SUBAPPLICATION Uebung_038 (* Lauflicht 8 reine Zeitsteuerung *)
  (* Standard: 61499-2; Description: Copyright (c) 2023 Meisterschulen am Ostbahnhof This program and the accompanying materials are made available under the terms of the Eclipse Public License 2.0 which is available at https://www.eclipse.org/legal/epl-2.0/ SPDX-License-Identifier: EPL-2.0 *)
  (* Version 1.0, 2023-10-23, Franz Höpfinger, Meisterschulen am Ostbahnhof *)
  PACKAGE Uebungen;
  IMPORT Uebungen::const::UT::DefaultPool::OutputNumber_N1;
  IMPORT logiBUS::io::DI::logiBUS_DI::Input_I1;
  IMPORT logiBUS::io::DI::logiBUS_DI::Input_I4;
  IMPORT logiBUS::io::DI::logiBUS_DI_Events::BUTTON_SINGLE_CLICK;
  IMPORT logiBUS::io::DQ::logiBUS_DO::Output_Q1;
  IMPORT logiBUS::io::DQ::logiBUS_DO::Output_Q2;
  IMPORT logiBUS::io::DQ::logiBUS_DO::Output_Q3;
  IMPORT logiBUS::io::DQ::logiBUS_DO::Output_Q4;
  IMPORT logiBUS::io::DQ::logiBUS_DO::Output_Q5;
  IMPORT logiBUS::io::DQ::logiBUS_DO::Output_Q6;
  IMPORT logiBUS::io::DQ::logiBUS_DO::Output_Q7;
  IMPORT logiBUS::io::DQ::logiBUS_DO::Output_Q8;
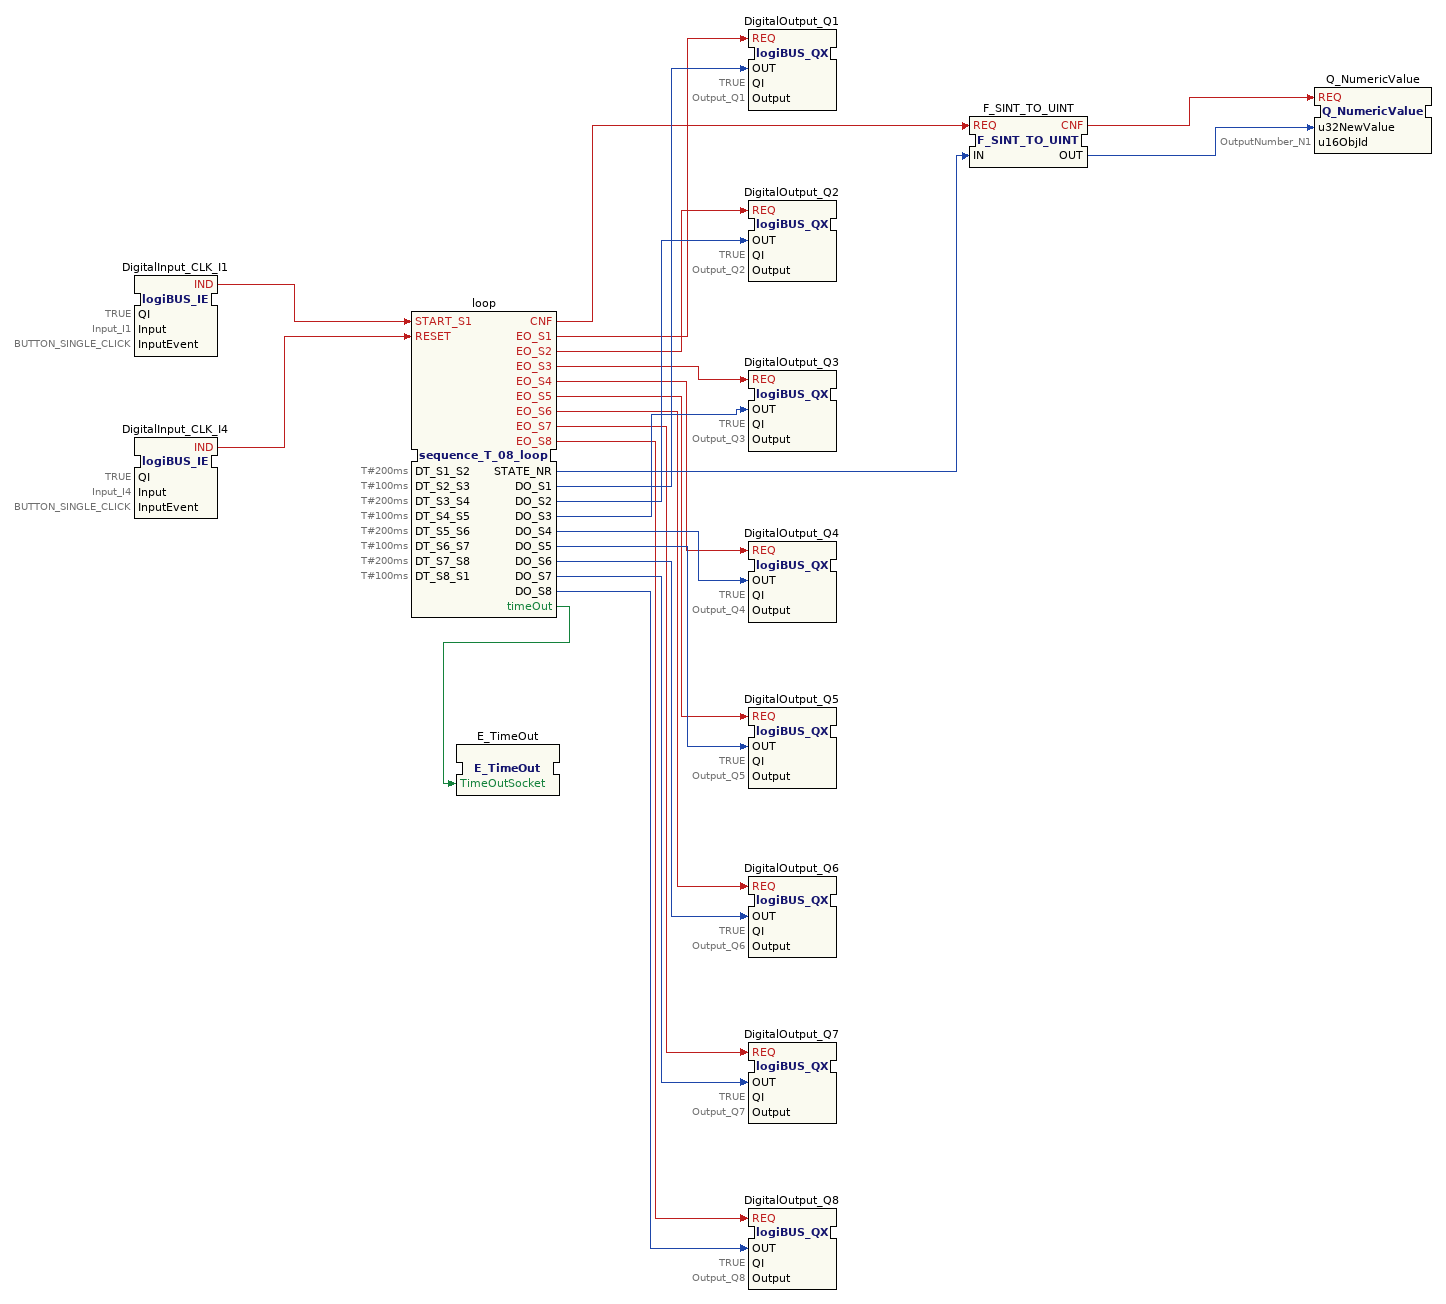
  FBS
    DigitalOutput_Q1 : logiBUS::io::DQ::logiBUS_QX(QI := TRUE, Output := Output_Q1);
    E_TimeOut : iec61499::events::E_TimeOut;
    DigitalOutput_Q2 : logiBUS::io::DQ::logiBUS_QX(QI := TRUE, Output := Output_Q2);
    DigitalOutput_Q3 : logiBUS::io::DQ::logiBUS_QX(QI := TRUE, Output := Output_Q3);
    DigitalOutput_Q4 : logiBUS::io::DQ::logiBUS_QX(QI := TRUE, Output := Output_Q4);
    DigitalInput_CLK_I1 : logiBUS::io::DI::logiBUS_IE(QI := TRUE, Input := Input_I1, InputEvent := BUTTON_SINGLE_CLICK);
    DigitalInput_CLK_I4 : logiBUS::io::DI::logiBUS_IE(QI := TRUE, Input := Input_I4, InputEvent := BUTTON_SINGLE_CLICK);
    DigitalOutput_Q5 : logiBUS::io::DQ::logiBUS_QX(QI := TRUE, Output := Output_Q5);
    DigitalOutput_Q6 : logiBUS::io::DQ::logiBUS_QX(QI := TRUE, Output := Output_Q6);
    DigitalOutput_Q7 : logiBUS::io::DQ::logiBUS_QX(QI := TRUE, Output := Output_Q7);
    DigitalOutput_Q8 : logiBUS::io::DQ::logiBUS_QX(QI := TRUE, Output := Output_Q8);
    Q_NumericValue : isobus::UT::Q::Q_NumericValue(u16ObjId := OutputNumber_N1);
    F_SINT_TO_UINT : iec61131::conversion::F_SINT_TO_UINT;
    loop : logiBUS::utils::sequence::timed::sequence_T_08_loop(DT_S1_S2 := T#200ms, DT_S2_S3 := T#100ms, DT_S3_S4 := T#200ms, DT_S4_S5 := T#100ms, DT_S5_S6 := T#200ms, DT_S6_S7 := T#100ms, DT_S7_S8 := T#200ms, DT_S8_S1 := T#100ms);
  END_FBS
  EVENT_CONNECTIONS
    F_SINT_TO_UINT.CNF TO Q_NumericValue.REQ;
    DigitalInput_CLK_I1.IND TO loop.START_S1;
    DigitalInput_CLK_I4.IND TO loop.RESET;
    loop.CNF TO F_SINT_TO_UINT.REQ;
    loop.EO_S1 TO DigitalOutput_Q1.REQ;
    loop.EO_S2 TO DigitalOutput_Q2.REQ;
    loop.EO_S3 TO DigitalOutput_Q3.REQ;
    loop.EO_S4 TO DigitalOutput_Q4.REQ;
    loop.EO_S5 TO DigitalOutput_Q5.REQ;
    loop.EO_S6 TO DigitalOutput_Q6.REQ;
    loop.EO_S7 TO DigitalOutput_Q7.REQ;
    loop.EO_S8 TO DigitalOutput_Q8.REQ;
  END_CONNECTIONS
  DATA_CONNECTIONS
    F_SINT_TO_UINT.OUT TO Q_NumericValue.u32NewValue;
    loop.STATE_NR TO F_SINT_TO_UINT.IN;
    loop.DO_S1 TO DigitalOutput_Q1.OUT;
    loop.DO_S2 TO DigitalOutput_Q2.OUT;
    loop.DO_S3 TO DigitalOutput_Q3.OUT;
    loop.DO_S4 TO DigitalOutput_Q4.OUT;
    loop.DO_S5 TO DigitalOutput_Q5.OUT;
    loop.DO_S6 TO DigitalOutput_Q6.OUT;
    loop.DO_S7 TO DigitalOutput_Q7.OUT;
    loop.DO_S8 TO DigitalOutput_Q8.OUT;
  END_CONNECTIONS
  ADAPTER_CONNECTIONS
    loop.timeOut TO E_TimeOut.TimeOutSocket;
  END_CONNECTIONS
END_SUBAPPLICATION
